PROGRAM INTERNAL _MAIN
VAR
END_VAR

END_PROGRAM

(* stored: Version 1.1.0.1, ProductVersion 3.1.4024.4
   POU _MAIN: Id {8e6ddbe0-2456-42a2-8b16-7085c8b833c4}, SpecialFunc None *)
